// TIA Portal V17 export
// export: Created 2024-08-07T21:44:13.079194Z, ExportSetting WithDefaults, DisplayName Totally Integrated Automation Portal, DisplayVersion V17 Update 7, DisplayName TIA Portal Openness, DisplayVersion V17 Update 7, DisplayName TIA Portal Version Control Interface, DisplayVersion V17, DisplayName SINAMICS Startdrive Advanced, DisplayVersion V17 SP2, DisplayName SINAMICS Startdrive G110M, G120, G120C, G120D, G120P, G115D, DisplayVersion V17 SP2, DisplayName SINAMICS Startdrive G130, G150, S120, S150, SINAMICS MV, S210, DisplayVersion V17 SP2, DisplayName STEP 7 Professional, DisplayVersion V17 Update 7, DisplayName STEP 7 Safety, DisplayVersion V17 Update 6, DisplayName WinCC Advanced / Unified PC, DisplayVersion V17 Update 7
VAR_GLOBAL   // PLC tag table "Cylinders_generated"
   iMM2200Bp__GrippingTubeFront AT %I21.0 : Bool;
   iMM2200Wp__GrippingTubeFront AT %I21.1 : Bool;
   qMM2200Bp__GrippingTubeFront AT %Q21.7 : Bool;
   qMM2200Wp__GrippingTubeFront AT %Q21.6 : Bool;
   iMM2201Bp__GrippingTubeRear AT %I21.2 : Bool;
   iMM2201Wp__GrippingTubeRear AT %I21.3 : Bool;
   iMM2220Bp__HoldingSidememberInsideLeft AT %I20.4 : Bool;
   iMM2220Wp__HoldingSidememberInsideLeft AT %I20.5 : Bool;
   qMM2220Bp__HoldingSidememberInsideLeft AT %Q22.7 : Bool;
   qMM2220Wp__HoldingSidememberInsideLeft AT %Q22.6 : Bool;
   iMM2221Bp__HoldingSidememberInsideRight AT %I20.6 : Bool;
   iMM2221Wp__HoldingSidememberInsideRight AT %I20.7 : Bool;
   iMM2240Bp__HoldingSidememberOutsideLeft AT %I20.0 : Bool;
   iMM2240Wp__HoldingSidememberOutsideLeft AT %I20.1 : Bool;
   qMM2240Bp__HoldingSidememberOutsideLeft AT %Q22.5 : Bool;
   qMM2240Wp__HoldingSidememberOutsideLeft AT %Q22.4 : Bool;
   iMM2241Bp__HoldingSidememberOutsideRight AT %I20.2 : Bool;
   iMM2241Wp__HoldingSidememberOutsideRight AT %I20.3 : Bool;
   iMM2500Bp__GrippingTubeFront AT %I24.0 : Bool;
   iMM2500Wp__GrippingTubeFront AT %I24.1 : Bool;
   qMM2500Bp__GrippingTubeFront AT %Q24.7 : Bool;
   qMM2500Wp__GrippingTubeFront AT %Q24.6 : Bool;
   iMM2501Bp__GrippingTubeRear AT %I24.2 : Bool;
   iMM2501Wp__GrippingTubeRear AT %I24.3 : Bool;
   iMM2520Bp__HoldingSidememberInsideLeft AT %I23.4 : Bool;
   iMM2520Wp__HoldingSidememberInsideLeft AT %I23.5 : Bool;
   qMM2520Bp__HoldingSidememberInsideLeft AT %Q25.7 : Bool;
   qMM2520Wp__HoldingSidememberInsideLeft AT %Q25.6 : Bool;
   iMM2521Bp__HoldingSidememberInsideRight AT %I23.6 : Bool;
   iMM2521Wp__HoldingSidememberInsideRight AT %I23.7 : Bool;
   iMM2540Bp__HoldingSidememberOutsideLeft AT %I23.0 : Bool;
   iMM2540Wp__HoldingSidememberOutsideLeft AT %I23.1 : Bool;
   qMM2540Bp__HoldingSidememberOutsideLeft AT %Q25.5 : Bool;
   qMM2540Wp__HoldingSidememberOutsideLeft AT %Q25.4 : Bool;
   iMM2541Bp__HoldingSidememberOutsideRight AT %I23.2 : Bool;
   iMM2541Wp__HoldingSidememberOutsideRight AT %I23.3 : Bool;
   iMM300Bp__ShiftingSupportRight AT %I25.0 : Bool;
   iMM300Wp__ShiftingSupportRight AT %I25.1 : Bool;
   qMM300Bp__ShiftingSupportRight AT %Q30.1 : Bool;
   qMM300Wp__ShiftingSupportRight AT %Q30.0 : Bool;
   iMM302Bp__ShiftingSupportLeft AT %I25.2 : Bool;
   iMM302Wp__ShiftingSupportLeft AT %I25.3 : Bool;
   qMM302Bp__ShiftingSupportLeft AT %Q30.3 : Bool;
   qMM302Wp__ShiftingSupportLeft AT %Q30.2 : Bool;
   iMM304Bp__MovingStopRight AT %I26.0 : Bool;
   iMM304Wp__MovingStopRight AT %I26.1 : Bool;
   qMM304Bp__MovingStopRight AT %Q30.5 : Bool;
   qMM304Wp__MovingStopRight AT %Q30.4 : Bool;
   iMM306Bp__MovingStopLeft AT %I26.2 : Bool;
   iMM306Wp__MovingStopLeft AT %I26.3 : Bool;
   qMM306Bp__MovingStopLeft AT %Q30.7 : Bool;
   qMM306Wp__MovingStopLeft AT %Q30.6 : Bool;
   iMM340Bp__RivetingUnitRight AT %I28.0 : Bool;
   iMM340Wp__RivetingUnitRight AT %I28.1 : Bool;
   qMM340Bp__RivetingUnitRight AT %Q34.1 : Bool;
   qMM340Wp__RivetingUnitRight AT %Q34.0 : Bool;
   iMM342Bp__RivetingUnitLeft AT %I28.2 : Bool;
   iMM342Wp__RivetingUnitLeft AT %I28.3 : Bool;
   qMM342Bp__RivetingUnitLeft AT %Q34.3 : Bool;
   qMM342Wp__RivetingUnitLeft AT %Q34.2 : Bool;
   iMM344Bp__RivetingSupportRight AT %I28.4 : Bool;
   iMM344Wp__RivetingSupportRight AT %I28.5 : Bool;
   qMM344Bp__RivetingSupportRight AT %Q34.5 : Bool;
   qMM344Wp__RivetingSupportRight AT %Q34.4 : Bool;
   iMM346Bp__RivetingSupportLeft AT %I28.6 : Bool;
   iMM346Wp__RivetingSupportLeft AT %I28.7 : Bool;
   qMM346Bp__RivetingSupportLeft AT %Q34.7 : Bool;
   qMM346Wp__RivetingSupportLeft AT %Q34.6 : Bool;
   iMM350Bp__ShiftWedgeRight AT %I25.6 : Bool;
   iMM350Wp__ShiftWedgeRight AT %I25.7 : Bool;
   qMM350Bp__ShiftWedgeRight AT %Q35.1 : Bool;
   qMM350Wp__ShiftWedgeRight AT %Q35.0 : Bool;
   iMM352Bp__ShiftWedgeLeft AT %I26.5 : Bool;
   iMM352Wp__ShiftWedgeLeft AT %I26.6 : Bool;
   qMM352Bp__ShiftWedgeLeft AT %Q35.3 : Bool;
   qMM352Wp__ShiftWedgeLeft AT %Q35.2 : Bool;
   iMM104Bp__AutoejectGripperLifting AT %I27.0 : Bool;
   iMM104Wp__AutoejectGripperLifting AT %I27.1 : Bool;
   qMM104Bp__AutoejectGripperLifting AT %Q10.5 : Bool;
   qMM104Wp__AutoejectGripperLifting AT %Q10.4 : Bool;
   iMM3100Bp__SidememberSupportLeft AT %I11.0 : Bool;
   iMM3100Wp__SidememberSupportLeft AT %I11.1 : Bool;
   qMM3100Bp__SidememberSupportLeft AT %Q31.1 : Bool;
   qMM3100Wp__SidememberSupportLeft AT %Q31.0 : Bool;
   iMM3101Bp__SidememberSupportRight AT %I11.2 : Bool;
   iMM3101Wp__SidememberSupportRight AT %I11.3 : Bool;
END_VAR
VAR_GLOBAL CONSTANT   // user constants
   NumberOfCylinders : Int := 25;
   MM2200_GrippingTubeFront : Int := 0;
   MM2201_GrippingTubeRear : Int := 1;
   MM2220_HoldingSidememberInsideLeft : Int := 2;
   MM2221_HoldingSidememberInsideRight : Int := 3;
   MM2240_HoldingSidememberOutsideLeft : Int := 4;
   MM2241_HoldingSidememberOutsideRight : Int := 5;
   MM2500_GrippingTubeFront : Int := 6;
   MM2501_GrippingTubeRear : Int := 7;
   MM2520_HoldingSidememberInsideLeft : Int := 8;
   MM2521_HoldingSidememberInsideRight : Int := 9;
   MM2540_HoldingSidememberOutsideLeft : Int := 10;
   MM2541_HoldingSidememberOutsideRight : Int := 11;
   MM300_ShiftingSupportRight : Int := 12;
   MM302_ShiftingSupportLeft : Int := 13;
   MM304_MovingStopRight : Int := 14;
   MM306_MovingStopLeft : Int := 15;
   MM340_RivetingUnitRight : Int := 16;
   MM342_RivetingUnitLeft : Int := 17;
   MM344_RivetingSupportRight : Int := 18;
   MM346_RivetingSupportLeft : Int := 19;
   MM350_ShiftWedgeRight : Int := 20;
   MM352_ShiftWedgeLeft : Int := 21;
   MM104_AutoejectGripperLifting : Int := 22;
   MM3100_SidememberSupport : Int := 23;
   MM3101_SidememberSupport : Int := 24;
END_VAR
